Fanuc KAREL source: IO0074.KL

-- PROVISIONAL review KL for V770-1; original PC SHA256 d09f670819710c4a9faad8e930c6e1d5a3a4b6dbb6a48992700924d88856f7c3
-- Incomplete behavior may be omitted. Consult companion uncertainty JSON. Do not deploy.
PROGRAM IO0074
%NOLOCKGROUP
-- UNRESOLVED_LOCAL_POOL 5 cells at code offset 13; source declarations unknown
-- DIRECT_LOCAL_WORD_ACCESS alone does not prove INTEGER, REAL, or BOOLEAN
BEGIN
  -- UNRESOLVED_PC offsets 0-18; opcodes 2B,2C,7B
  -- UNRESOLVED_PC offsets 23-30; opcodes 9D,23
  -- UNRESOLVED_PC offsets 35-49; opcodes 2E,22,9D,33,35
  -- UNRESOLVED_PC offsets 54-61; opcodes 9D,23
  -- UNRESOLVED_PC offsets 66-77; opcodes 2E,23
  -- UNRESOLVED_PC offsets 82-105; opcodes 22,21,33,34,19,64,23
  -- UNRESOLVED_PC offsets 110-114; opcodes 7F
  -- UNRESOLVED_PC offsets 119-123; opcodes 27,AA
  -- UNRESOLVED_PC offsets 128-132; opcodes 7F
END IO0074
